// TIA Portal project "KPB" (V19)
// prva verzija - pokusaj izrade hominga

(* hardware
DEVICE "S7-1200 station_1"  S7-1200 Station
   slot 0: "Rack_0"  S7-1200 Rack  Rack  V1.0
   slot 1: "PLC_1"  CPU 1215C DC/DC/DC  6ES7 215-1AG40-0XB0  V4.0
*)

// ===== PLC "PLC_1"  CPU 1215C DC/DC/DC =====

VAR_GLOBAL   // PLC tag table "Default tag table"
   "spustanje" AT %I0.5 : Bool;
   "m_spustanje" AT %M0.2 : Bool;
   "podizanje" AT %I0.4 : Bool;
   "m_podizanje" AT %M0.3 : Bool;
   "reset" AT %M0.4 : Bool;
   "Mikroprekidac_homing" AT %I1.0 : Bool;
   "pneumatski razvodnik" AT %Q0.3 : Bool;
   "broj_pritisaka_paran" AT %M0.5 : Bool;
   "broj_pritisaka" AT %M0.6 : Bool;
   "Disconnect" AT %M2.1 : Bool;
   "Send_data" AT %M2.3 : Bool;
   "Connection_established" AT %M2.2 : Bool;
END_VAR

VAR_GLOBAL   // PLC tag table "Koracni_motor"
   "pulse" AT %Q0.2 : Bool;   // crna zica
   "enable" AT %Q0.1 : Bool;   // smedja zica
   "direction" AT %Q0.0 : Bool;   // bijela zica
   "Gljiva" AT %I0.0 : Bool;
   "povecanje_brzine" AT %I0.6 : Bool;
   "smanjenje_brzine" AT %I0.7 : Bool;
   "m_povecanje" AT %M0.0 : Bool;
   "m_smanjenje" AT %M0.1 : Bool;
END_VAR

VAR_GLOBAL   // PLC tag table "Homing"
   "Mikroprekidac_G" AT %I0.1 : Bool;   // gornji hw
   "Mikroprekidac_D" AT %I0.2 : Bool;   // donji hw
   "busenje" AT %I0.3 : Bool;
END_VAR

VAR_GLOBAL   // PLC tag table "komunikacija"
   "connect" AT %M2.0 : Bool;
END_VAR

VAR_GLOBAL   // PLC tag table "konstantna_pb"
   "pokreni" AT %M3.0 : Bool;
   "busenje_u_tijeku" AT %M3.1 : Bool;
   "stop" AT %M3.2 : Bool;
END_VAR

VAR_GLOBAL   // PLC tag table "Clock Memory"
   "Clock_Byte" AT %MB100 : Byte;
   "Clock_10Hz" AT %M100.0 : Bool;
   "Clock_5Hz" AT %M100.1 : Bool;
   "Clock_2.5Hz" AT %M100.2 : Bool;
   "Clock_2Hz" AT %M100.3 : Bool;
   "Clock_1.25Hz" AT %M100.4 : Bool;
   "Clock_1Hz" AT %M100.5 : Bool;
   "Clock_0.625Hz" AT %M100.6 : Bool;
   "Clock_0.5Hz" AT %M100.7 : Bool;
END_VAR

DATA_BLOCK "rucno_upravljanje"   // DB10
{ S7_Optimized_Access := 'TRUE' }
VERSION : 0.1
   VAR
      konstantna_brzina : Real := 1.0;
      brzina : Real := 8.0;
      broj_pritisaka : Int;
      homing : Bool;
      set_reset : Bool;
      h2 : Bool;
      rezultat : Int;
   END_VAR
BEGIN
END_DATA_BLOCK

DATA_BLOCK "Receive_here"   // DB13
{ S7_Optimized_Access := 'FALSE' }
VERSION : 0.1
   VAR
      Z_Sila : Real;
   END_VAR
BEGIN
END_DATA_BLOCK

DATA_BLOCK "Bušenje_ON"   // DB15
{ S7_Optimized_Access := 'FALSE' }
VERSION : 0.1
   VAR
      bON : Bool := true;
   END_VAR
BEGIN
END_DATA_BLOCK

DATA_BLOCK "detekcija_proboja"   // DB18
{ S7_Optimized_Access := 'TRUE' }
VERSION : 0.1
   VAR
      prag_vrijednosti_sile : Real := 20.0;
      sloj1 : Bool;
      sloj2 : Bool;
      sloj3 : Bool;
      zavrsetak : Bool;
      proboj : Bool;
   END_VAR
BEGIN
END_DATA_BLOCK

DATA_BLOCK "Bušenje_OFF"   // DB20
{ S7_Optimized_Access := 'FALSE' }
VERSION : 0.1
   VAR
      bOFF : Bool;
   END_VAR
BEGIN
END_DATA_BLOCK

DATA_BLOCK "Pomocni_blok"   // DB30
{ S7_Optimized_Access := 'TRUE' }
VERSION : 0.1
   VAR
      "100Hz" : Bool;
      Posalji_ON : Bool;
      Posalji_OFF : Bool;
   END_VAR
BEGIN
END_DATA_BLOCK

DATA_BLOCK "PB"   // DB31
{ S7_Optimized_Access := 'FALSE' }
VERSION : 0.1
   VAR
      PB : Real := 1.0;
   END_VAR
BEGIN
END_DATA_BLOCK

// folder: System blocks/Program resources

DATA_BLOCK "IEC_Timer_0_DB"   // DB7
{ S7_Optimized_Access := 'TRUE' }
AUTHOR : Simatic
FAMILY : IEC
NAME : IEC_TMR
VERSION : 1.0
// stored: InstanceOfName IEC_TIMER
"IEC_TIMER"
BEGIN
END_DATA_BLOCK

DATA_BLOCK "PLC_1_Connection_DB"   // DB9
{ S7_Optimized_Access := 'TRUE' }
AUTHOR : SIMATIC
FAMILY : MC7Plus
NAME : TCON_Prm
VERSION : 1.0
// stored: InstanceOfName TCON_Param
"TCON_Param"
BEGIN
   ID := 1;
   REM_TSAP_ID_LEN := 0;
   LOCAL_TSAP_ID[1] := B#16#07;
   LOCAL_TSAP_ID[2] := B#16#D0;
   LOCAL_TSAP_ID_LEN := 2;
   ACTIVE_EST := false;
   REM_STADDR[1] := 192;
   REM_STADDR[2] := 168;
   REM_STADDR[4] := 241;
END_DATA_BLOCK

DATA_BLOCK "IEC_Timer_0_DB_1"   // DB19
{ S7_Optimized_Access := 'TRUE' }
AUTHOR : Simatic
FAMILY : IEC
NAME : IEC_TMR
VERSION : 1.0
// stored: InstanceOfName IEC_TIMER
"IEC_TIMER"
BEGIN
END_DATA_BLOCK

DATA_BLOCK "IEC_Timer_0_DB_3"   // DB22
{ S7_Optimized_Access := 'TRUE' }
AUTHOR : Simatic
FAMILY : IEC
NAME : IEC_TMR
VERSION : 1.0
// stored: InstanceOfName IEC_TIMER
"IEC_TIMER"
BEGIN
END_DATA_BLOCK

DATA_BLOCK "IEC_Timer_0_DB_2"   // DB23
{ S7_Optimized_Access := 'TRUE' }
AUTHOR : Simatic
FAMILY : IEC
NAME : IEC_TMR
VERSION : 1.0
// stored: InstanceOfName IEC_TIMER
"IEC_TIMER"
BEGIN
END_DATA_BLOCK

DATA_BLOCK "IEC_Timer_0_DB_7"   // DB26
{ S7_Optimized_Access := 'TRUE' }
AUTHOR : Simatic
FAMILY : IEC
NAME : IEC_TMR
VERSION : 1.0
// stored: InstanceOfName IEC_TIMER
"IEC_TIMER"
BEGIN
END_DATA_BLOCK

DATA_BLOCK "IEC_Timer_0_DB_5"   // DB28
{ S7_Optimized_Access := 'TRUE' }
AUTHOR : Simatic
FAMILY : IEC
NAME : IEC_TMR
VERSION : 1.0
// stored: InstanceOfName IEC_TIMER
"IEC_TIMER"
BEGIN
END_DATA_BLOCK

DATA_BLOCK "IEC_Timer_0_DB_8"   // DB29
{ S7_Optimized_Access := 'TRUE' }
AUTHOR : Simatic
FAMILY : IEC
NAME : IEC_TMR
VERSION : 1.0
// stored: InstanceOfName IEC_TIMER
"IEC_TIMER"
BEGIN
END_DATA_BLOCK

// folder: (top level)

DATA_BLOCK "Axis"   // DB2, Motion_DB
{ S7_Optimized_Access := 'TRUE' }
AUTHOR : SIMATIC
FAMILY : BasicMC
NAME : TO_PosAx
VERSION : 4.0
// stored: InstanceOfName TO_PositioningAxis
"TO_PositioningAxis"
BEGIN
   // Axis.HomingReferencePointSwitch_AddressCU = %I1.0
   // Axis.LengthUnitNormalized.Distance = 1013
   // Axis.PositionLimitsMax_AddressCU = %I0.2
   // Axis.PositionLimitsMin_AddressCU = %I0.1
   // Axis.EnableOutput_AddressCU = %Q0.1
   // Axis.OnlinePtoModeCU = 16#0000_0002
   // Axis.DirectionOutputEnabledCU = TRUE
   // Axis.SelectedChannel2EnumCU = %Q0.0
   // Axis.SelectedChannel1EnumCU = %Q0.2
   // Pulse.MinDeltaDeltaFrequencyCU = 0.004
   // Pulse.MaxDeltaDeltaFrequencyCU = 1.0E+10
   // Pulse.MinDeltaFrequencyCU = 0.005
   // Pulse.MaxDeltaFrequencyCU = 9.5E+9
   // Pulse.MinFrequencyCU = 1.0
   // Pulse.MaxFrequencyCU = 100000.0
   // Pulse.OutputSourceCU = 16#0000_0000
   // Axis.SelectPTO = 0
END_DATA_BLOCK

FUNCTION "FC_proboj" : Void   // FC1, LAD
{ S7_Optimized_Access := 'TRUE' }
VERSION : 0.1
   VAR_TEMP   // added for the SCL form of the ladder/FBD networks
      _w1 : Bool;
   END_VAR
BEGIN

REGION Network 1
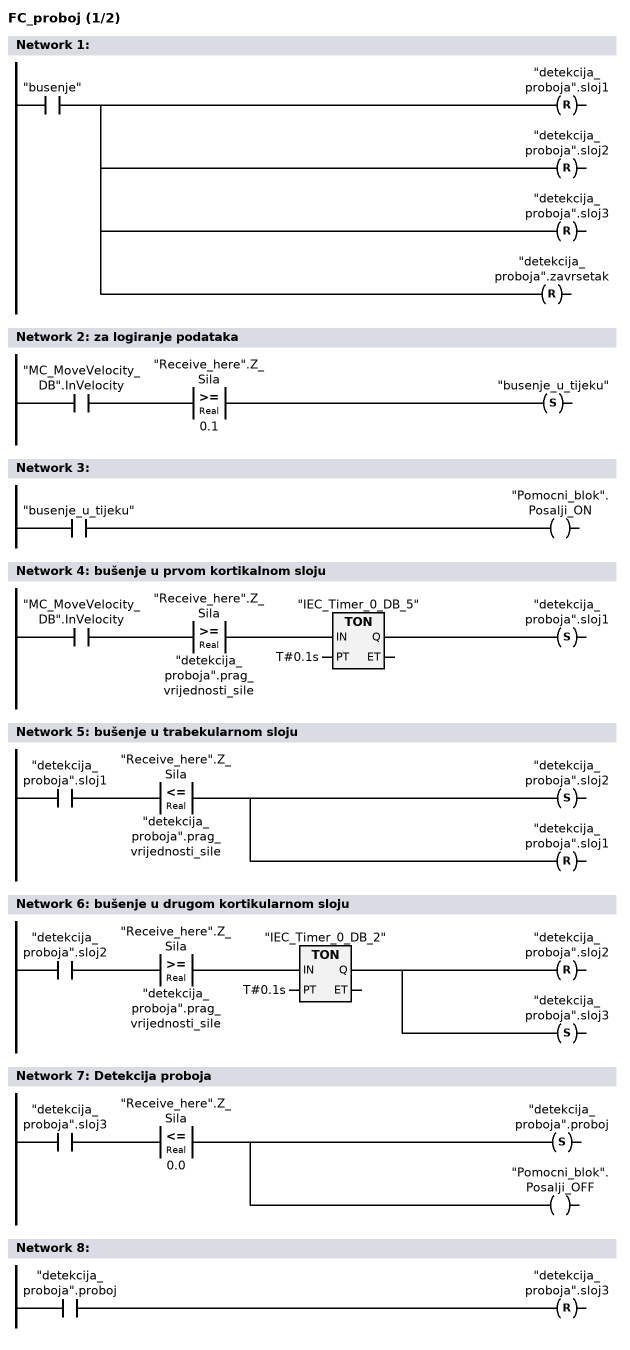
   RUNG wire#powerrail
      Contact( "busenje" )
      wire#w1
      R_Coil( "detekcija_proboja".sloj1 )
   END_RUNG
   RUNG wire#w1
      R_Coil( "detekcija_proboja".sloj2 )
   END_RUNG
   RUNG wire#w1
      R_Coil( "detekcija_proboja".sloj3 )
   END_RUNG
   RUNG wire#w1
      R_Coil( "detekcija_proboja".zavrsetak )
   END_RUNG
   // the same network as SCL:
   IF "busenje" THEN
       "detekcija_proboja".sloj1 := FALSE;
       "detekcija_proboja".sloj2 := FALSE;
       "detekcija_proboja".sloj3 := FALSE;
       "detekcija_proboja".zavrsetak := FALSE;
   END_IF;
END_REGION

REGION Network 2: za logiranje podataka
   RUNG wire#powerrail
      Contact( "MC_MoveVelocity_DB".InVelocity )
      { S7_Templates := "SrcType := Real" } GE_Contact(in1 := "Receive_here".Z_Sila, in2 := 0.1)
      S_Coil( "busenje_u_tijeku" )
   END_RUNG
   // the same network as SCL:
   IF "MC_MoveVelocity_DB".InVelocity AND ("Receive_here".Z_Sila >= 0.1) THEN
       "busenje_u_tijeku" := TRUE;
   END_IF;
END_REGION

REGION Network 3
   RUNG wire#powerrail
      Contact( "busenje_u_tijeku" )
      Coil( "Pomocni_blok".Posalji_ON )
   END_RUNG
   // the same network as SCL:
   "Pomocni_blok".Posalji_ON := "busenje_u_tijeku";
END_REGION

REGION Network 4: bušenje u prvom kortikalnom sloju
   "IEC_Timer_0_DB_5".TON(IN := "MC_MoveVelocity_DB".InVelocity AND ("Receive_here".Z_Sila >= "detekcija_proboja".prag_vrijednosti_sile),
                          PT := T#0.1s);
   IF "IEC_Timer_0_DB_5".Q THEN "detekcija_proboja".sloj1 := TRUE; END_IF;
END_REGION

REGION Network 5: bušenje u trabekularnom sloju
   RUNG wire#powerrail
      Contact( "detekcija_proboja".sloj1 )
      { S7_Templates := "SrcType := Real" } LE_Contact(in1 := "Receive_here".Z_Sila, in2 := "detekcija_proboja".prag_vrijednosti_sile)
      wire#w1
      S_Coil( "detekcija_proboja".sloj2 )
   END_RUNG
   RUNG wire#w1
      R_Coil( "detekcija_proboja".sloj1 )
   END_RUNG
   // the same network as SCL:
   IF "detekcija_proboja".sloj1 AND ("Receive_here".Z_Sila <= "detekcija_proboja".prag_vrijednosti_sile) THEN
       "detekcija_proboja".sloj2 := TRUE;
       "detekcija_proboja".sloj1 := FALSE;
   END_IF;
END_REGION

REGION Network 6: bušenje u drugom kortikularnom sloju
   "IEC_Timer_0_DB_2".TON(IN := "detekcija_proboja".sloj2 AND ("Receive_here".Z_Sila >= "detekcija_proboja".prag_vrijednosti_sile),
                          PT := T#0.1s);
   IF "IEC_Timer_0_DB_2".Q THEN
       "detekcija_proboja".sloj2 := FALSE;
       "detekcija_proboja".sloj3 := TRUE;
   END_IF;
END_REGION

REGION Network 7: Detekcija proboja
   RUNG wire#powerrail
      Contact( "detekcija_proboja".sloj3 )
      { S7_Templates := "SrcType := Real" } LE_Contact(in1 := "Receive_here".Z_Sila, in2 := 0.0)
      wire#w1
      S_Coil( "detekcija_proboja".proboj )
   END_RUNG
   RUNG wire#w1
      Coil( "Pomocni_blok".Posalji_OFF )
   END_RUNG
   // the same network as SCL:
   #_w1 := "detekcija_proboja".sloj3 AND ("Receive_here".Z_Sila <= 0.0);
   IF #_w1 THEN "detekcija_proboja".proboj := TRUE; END_IF;
   "Pomocni_blok".Posalji_OFF := #_w1;
END_REGION

REGION Network 8
   RUNG wire#powerrail
      Contact( "detekcija_proboja".proboj )
      R_Coil( "detekcija_proboja".sloj3 )
   END_RUNG
   // the same network as SCL:
   IF "detekcija_proboja".proboj THEN "detekcija_proboja".sloj3 := FALSE; END_IF;
END_REGION

REGION Network 9
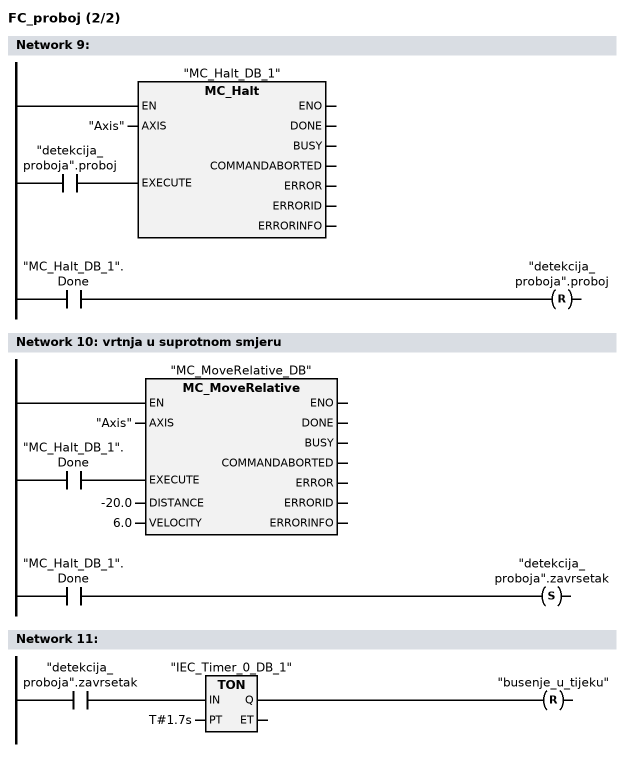
   "MC_Halt_DB_1"(Axis := "Axis", Execute := "detekcija_proboja".proboj);   // MC_Halt
   IF "MC_Halt_DB_1".Done THEN "detekcija_proboja".proboj := FALSE; END_IF;
END_REGION

REGION Network 10: vrtnja u suprotnom smjeru
   "MC_MoveRelative_DB"(Axis := "Axis", Execute := "MC_Halt_DB_1".Done, Distance := -20.0, Velocity := 6.0);   // MC_MoveRelative
   IF "MC_Halt_DB_1".Done THEN "detekcija_proboja".zavrsetak := TRUE; END_IF;
END_REGION

REGION Network 11
   "IEC_Timer_0_DB_1".TON(IN := "detekcija_proboja".zavrsetak, PT := T#1.7s);
   IF "IEC_Timer_0_DB_1".Q THEN "busenje_u_tijeku" := FALSE; END_IF;
END_REGION
END_FUNCTION

FUNCTION "TCP_ON_OFF" : Void   // FC2, LAD
{ S7_Optimized_Access := 'TRUE' }
VERSION : 0.1
BEGIN

REGION Network 1: komunikacija TCON
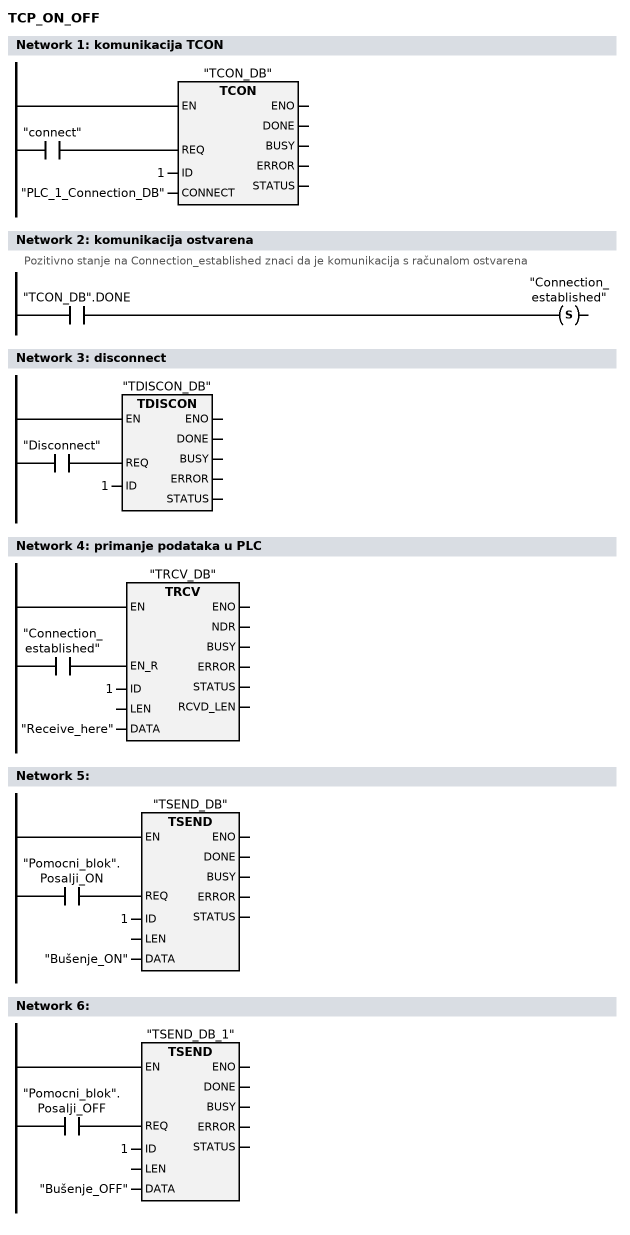
   "TCON_DB"(REQ := "connect", ID := 1, CONNECT := "PLC_1_Connection_DB");   // TCON
END_REGION

REGION Network 2: komunikacija ostvarena
   // Pozitivno stanje na Connection_established znaci da je komunikacija s računalom ostvarena
   RUNG wire#powerrail
      Contact( "TCON_DB".DONE )
      S_Coil( "Connection_established" )
   END_RUNG
   // the same network as SCL:
   IF "TCON_DB".DONE THEN "Connection_established" := TRUE; END_IF;
END_REGION

REGION Network 3: disconnect
   "TDISCON_DB"(REQ := "Disconnect", ID := 1);   // TDISCON
END_REGION

REGION Network 4: primanje podataka u PLC
   "TRCV_DB"(EN_R := "Connection_established", ID := 1, DATA := "Receive_here");   // TRCV
END_REGION

REGION Network 5
   "TSEND_DB"(REQ := "Pomocni_blok".Posalji_ON, ID := 1, DATA := "Bušenje_ON");   // TSEND
END_REGION

REGION Network 6
   "TSEND_DB_1"(REQ := "Pomocni_blok".Posalji_OFF, ID := 1, DATA := "Bušenje_OFF");   // TSEND
END_REGION
END_FUNCTION

FUNCTION "Logiranje" : Void   // FC4, LAD
{ S7_Optimized_Access := 'TRUE' }
VERSION : 0.1
BEGIN

REGION Network 1: logiranje vrijednosti sile frekvencijom od 100 Hz
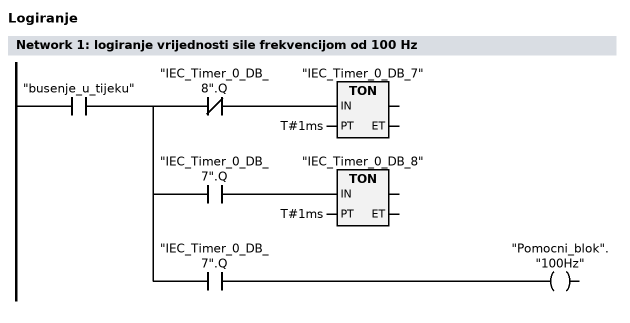
   "IEC_Timer_0_DB_7".TON(IN := "busenje_u_tijeku" AND NOT "IEC_Timer_0_DB_8".Q, PT := T#1ms);
   "IEC_Timer_0_DB_8".TON(IN := "busenje_u_tijeku" AND "IEC_Timer_0_DB_7".Q, PT := T#1ms);
   "Pomocni_blok"."100Hz" := "busenje_u_tijeku" AND "IEC_Timer_0_DB_7".Q;
END_REGION
END_FUNCTION

ORGANIZATION_BLOCK "upravljanje"   // OB123, LAD, ProgramCycle
TITLE = "Main Program Sweep (Cycle)"
{ S7_Optimized_Access := 'TRUE' }
VERSION : 0.1
   VAR_INPUT
      Initial_Call : Bool;   // Initial call of this OB
      Remanence : Bool;   // =True, if remanent data are available
   END_VAR
   VAR_TEMP   // added for the SCL form of the ladder/FBD networks
      _w1 : Bool;
      _w2 : Bool;
      _w3 : Bool;
      _w4 : Bool;
   END_VAR
BEGIN

REGION Network 1: power
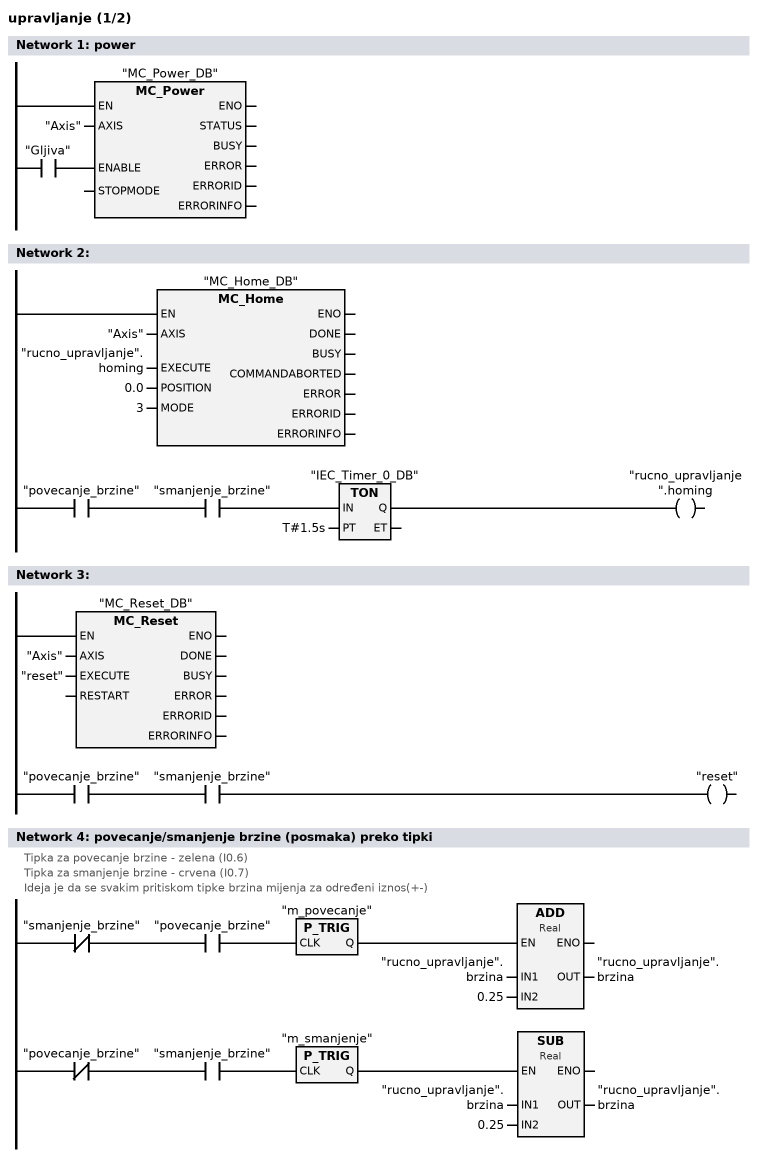
   "MC_Power_DB"(Axis := "Axis", Enable := "Gljiva");   // MC_Power
END_REGION

REGION Network 2
   "MC_Home_DB"(Axis := "Axis", Execute := "rucno_upravljanje".homing, Position := 0.0, Mode := 3);   // MC_Home
   "IEC_Timer_0_DB".TON(IN := "povecanje_brzine" AND "smanjenje_brzine", PT := T#1.5s);
   "rucno_upravljanje".homing := "IEC_Timer_0_DB".Q;
END_REGION

REGION Network 3
   "MC_Reset_DB"(Axis := "Axis", Execute := "reset");   // MC_Reset
   "reset" := "povecanje_brzine" AND "smanjenje_brzine";
END_REGION

REGION Network 4: povecanje/smanjenje brzine (posmaka) preko tipki
   // Tipka za povecanje brzine - zelena (I0.6)
   // Tipka za smanjenje brzine - crvena (I0.7)
   // Ideja je da se svakim pritiskom tipke brzina mijenja za određeni iznos(+-)
   RUNG wire#powerrail
      I_Contact( "smanjenje_brzine" )
      Contact( "povecanje_brzine" )
      P_Trig( "m_povecanje" )
      { S7_Templates := "SrcType := Real" } Add(in1 := "rucno_upravljanje".brzina, in2 := 0.25, out => "rucno_upravljanje".brzina)
   END_RUNG
   RUNG wire#powerrail
      I_Contact( "povecanje_brzine" )
      Contact( "smanjenje_brzine" )
      P_Trig( "m_smanjenje" )
      { S7_Templates := "SrcType := Real" } Sub(in1 := "rucno_upravljanje".brzina, in2 := 0.25, out => "rucno_upravljanje".brzina)
   END_RUNG
   // the same network as SCL:
   #_w1 := NOT "smanjenje_brzine" AND "povecanje_brzine";
   #_w2 := #_w1 AND NOT "m_povecanje";   // rising edge
   "m_povecanje" := #_w1;
   IF #_w2 THEN "rucno_upravljanje".brzina := "rucno_upravljanje".brzina + 0.25; END_IF;
   #_w3 := NOT "povecanje_brzine" AND "smanjenje_brzine";
   #_w4 := #_w3 AND NOT "m_smanjenje";   // rising edge
   "m_smanjenje" := #_w3;
   IF #_w4 THEN "rucno_upravljanje".brzina := "rucno_upravljanje".brzina - 0.25; END_IF;
END_REGION

REGION Network 5: rucno podizanje i spustanje
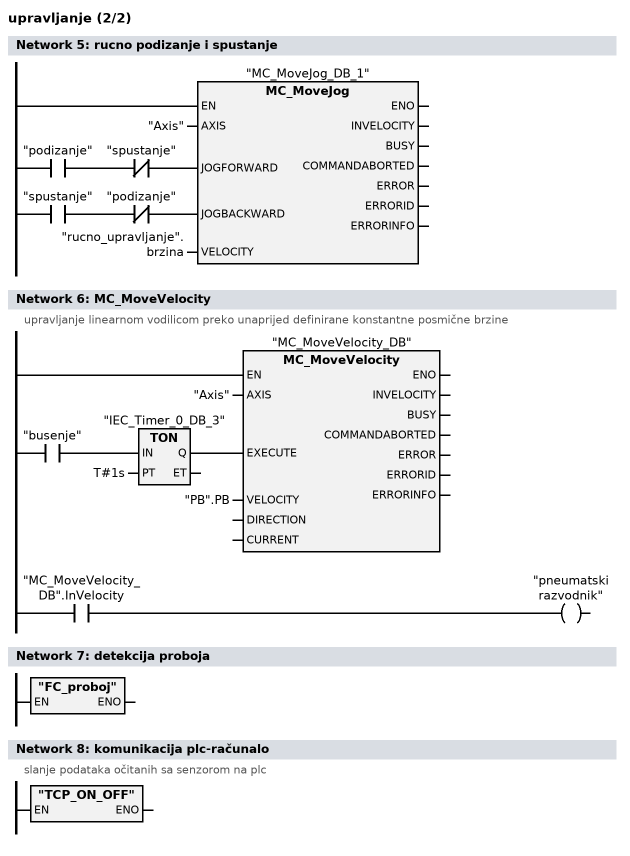
   "MC_MoveJog_DB_1"(Axis := "Axis",   // MC_MoveJog
                     JogForward := "podizanje" AND NOT "spustanje",
                     JogBackward := "spustanje" AND NOT "podizanje",
                     Velocity := "rucno_upravljanje".brzina);
END_REGION

REGION Network 6: MC_MoveVelocity
   // upravljanje linearnom vodilicom preko unaprijed definirane konstantne posmične brzine
   "IEC_Timer_0_DB_3".TON(IN := "busenje", PT := T#1s);
   "MC_MoveVelocity_DB"(Axis := "Axis", Execute := "IEC_Timer_0_DB_3".Q, Velocity := "PB".PB);   // MC_MoveVelocity
   "pneumatski razvodnik" := "MC_MoveVelocity_DB".InVelocity;
END_REGION

REGION Network 7: detekcija proboja
   RUNG wire#powerrail
      "FC_proboj"()
   END_RUNG
   // the same network as SCL:
   "FC_proboj"();
END_REGION

REGION Network 8: komunikacija plc-računalo
   // slanje podataka očitanih sa senzorom na plc
   RUNG wire#powerrail
      "TCP_ON_OFF"()
   END_RUNG
   // the same network as SCL:
   "TCP_ON_OFF"();
END_REGION
END_ORGANIZATION_BLOCK